// Mitsubishi GX Works2 project: automation_group14_plc_280124   PLC: FX3G

// global labels: Global1
VAR_GLOBAL
  start AT X007 : BOOL;
  During_day AT Y007 : BOOL;
  Emergency_B AT X011 : BOOL;
  Analog_Input1 AT D8280 : INT;
  input_value AT D8201 : INT;
END_VAR
VAR_GLOBAL CONSTANT
  less_then_5 : REAL;
  check_if_lager : INT := 5;
END_VAR
VAR_GLOBAL
  Lager AT M2 : BOOL;
  On_Switch AT X007 : BOOL;
  analog_output AT D8282 : INT;
  check_inv AT M1 : BOOL;
  Analog_Value1 AT D8288 : INT;
END_VAR
VAR_GLOBAL CONSTANT
  Middle_Val : REAL := 2000;
END_VAR
VAR_GLOBAL
  Beer_Type AT M2 : BOOL;
  enough_inv AT M3 : BOOL;
  check AT Y000 : BOOL;
  Input_val AT D8280 : REAL;
END_VAR
VAR_GLOBAL CONSTANT
  div_by_400 : INT := 400;
END_VAR
VAR_GLOBAL
  save_Analog_V AT D7777 : REAL;
END_VAR
VAR_GLOBAL CONSTANT
  normalization : REAL := 400;
END_VAR
VAR_GLOBAL
  option AT D2000 : REAL;
END_VAR
VAR_GLOBAL CONSTANT
  const_1 : REAL := 5;
END_VAR
VAR_GLOBAL
  inv_good AT M3 : BOOL;
  TC_1 AT Y001 : BOOL;
  TC AT TC1 : BOOL;
END_VAR
VAR_GLOBAL CONSTANT
  timer_1 : REAL := 40;
END_VAR
VAR_GLOBAL
  timer_when_cooking AT TS1 : BOOL;
  y_1 AT Y001 : BOOL;
  TC1 AT TC1 : BOOL;
END_VAR
VAR_GLOBAL CONSTANT
  TIMER_COOKING : INT := 40;
END_VAR
VAR_GLOBAL
  job_1 AT X001 : BOOL;
  lagger_check AT M4 : BOOL;
  pilzner_check AT M5 : BOOL;
END_VAR
VAR_GLOBAL CONSTANT
  Lager_Shmarim_need : REAL := 150;
  Lager_Letet_need : REAL := 12;
  Lager_Kshut_need : REAL := 60;
  Pilzner_Shmarim_need : REAL := 120;
  Pilzner_letet_need : REAL := 6;
  Pilzner_Kshut_need : REAL := 53;
  shmarim : REAL := 301;
  letet : REAL := 200;
  kshut : REAL := 200;
END_VAR
VAR_GLOBAL
  finished_cooking_lagger AT M6 : BOOL;
  shmarim_inv AT D4444 : REAL;
  letet_inv AT D5555 : REAL;
  kshut_inv AT D6666 : REAL;
  finished_cooking_Pilzner AT M7 : BOOL;
  move_to_tsisa AT X005 : BOOL;
  start_tsisa_lagger AT M8 : BOOL;
  start_tsisa_pilzner AT M9 : BOOL;
END_VAR
VAR_GLOBAL CONSTANT
  TValue3 : INT := 30;
END_VAR
VAR_GLOBAL
  TS1 AT TS1 : BOOL;
  Y_3 AT Y003 : BOOL;
  TC_4 AT TC4 : BOOL;
END_VAR
VAR_GLOBAL CONSTANT
  TValue4 : INT := 40;
END_VAR
VAR_GLOBAL
  TS_4 AT TS4 : BOOL;
  y_4 AT Y004 : BOOL;
  X_2 AT X002 : BOOL;
  X_0 AT X000 : BOOL;
  cc_1 AT CC1 : BOOL;
END_VAR
VAR_GLOBAL CONSTANT
  counter5 : INT := 6;
END_VAR
VAR_GLOBAL
  CS_1 AT CS1 : BOOL;
  Y_2 AT Y002 : BOOL;
  m_11 AT M11 : BOOL;
  TC_5 AT TC5 : BOOL;
  TS_5 AT TS5 : BOOL;
  TC_6 AT TC6 : BOOL;
  TS_6 AT TS6 : BOOL;
  m_20 AT M20 : BOOL;
  NumOfPack AT D1111 : REAL;
END_VAR
VAR_GLOBAL CONSTANT
  AddingPack : REAL := 0.1;
END_VAR
VAR_GLOBAL
  DayFinish_Lager AT M18 : BOOL;
  DayFinish_Pilzner AT M19 : BOOL;
END_VAR
VAR_GLOBAL CONSTANT
  MulFourty : REAL := 4000;
END_VAR
VAR_GLOBAL
  m_21 AT M21 : BOOL;
  is_Lager AT M2 : BOOL;
  is_pilzner AT M21 : BOOL;
END_VAR
VAR_GLOBAL CONSTANT
  counter6 : INT := 6;
END_VAR
VAR_GLOBAL
  X0_isOn AT M25 : BOOL;
  DayFinish AT M30 : BOOL;
  Not_day_finish AT M30 : BOOL;
END_VAR
VAR_GLOBAL CONSTANT
  const_2 : REAL := 10;
END_VAR
VAR_GLOBAL
  TC_3 AT TC3 : BOOL;
  TS_3 AT TS3 : BOOL;
  Not_finish_Pack_1 AT M40 : BOOL;
END_VAR
VAR_GLOBAL CONSTANT
  div_forty : REAL := 10;
END_VAR
VAR_GLOBAL
  final_output AT D6000 : REAL;
END_VAR
VAR_GLOBAL CONSTANT
  MulFourty1 : REAL := 10;
END_VAR
VAR_GLOBAL
  analog_output1 AT D8282 : INT;
  TC13 AT TC13 : BOOL;
  TsisaLager AT TC13 : BOOL;
END_VAR
VAR_GLOBAL CONSTANT
  tsisaLager_30 : INT := 30;
END_VAR
VAR_GLOBAL
  TsisaPilzner AT TC14 : BOOL;
END_VAR
VAR_GLOBAL CONSTANT
  tsisaPilzner_40 : INT := 40;
END_VAR
VAR_GLOBAL
  finish_tsia_lager AT TS13 : BOOL;
  finish_tsisa_pilzner AT TS14 : BOOL;
  M_100 AT M100 : BOOL;
  start_blink3 AT TC30 : BOOL;
END_VAR
VAR_GLOBAL CONSTANT
  Blink : INT := 5;
END_VAR
VAR_GLOBAL
  blink_Y3 AT TS30 : BOOL;
  start_blink4 AT TC31 : BOOL;
END_VAR
VAR_GLOBAL CONSTANT
  blink2 : INT := 5;
END_VAR
VAR_GLOBAL
  Blink_Y4 AT TS31 : BOOL;
END_VAR

// task Task_01 (event TRUE, interval 0, priority 31): POU_01

PROGRAM POU_01
(* structured ladder/FBD written out as ST: instructions are called as NAME(EN, inputs, outputs); _pN, _eN, _tN stand for wires *)
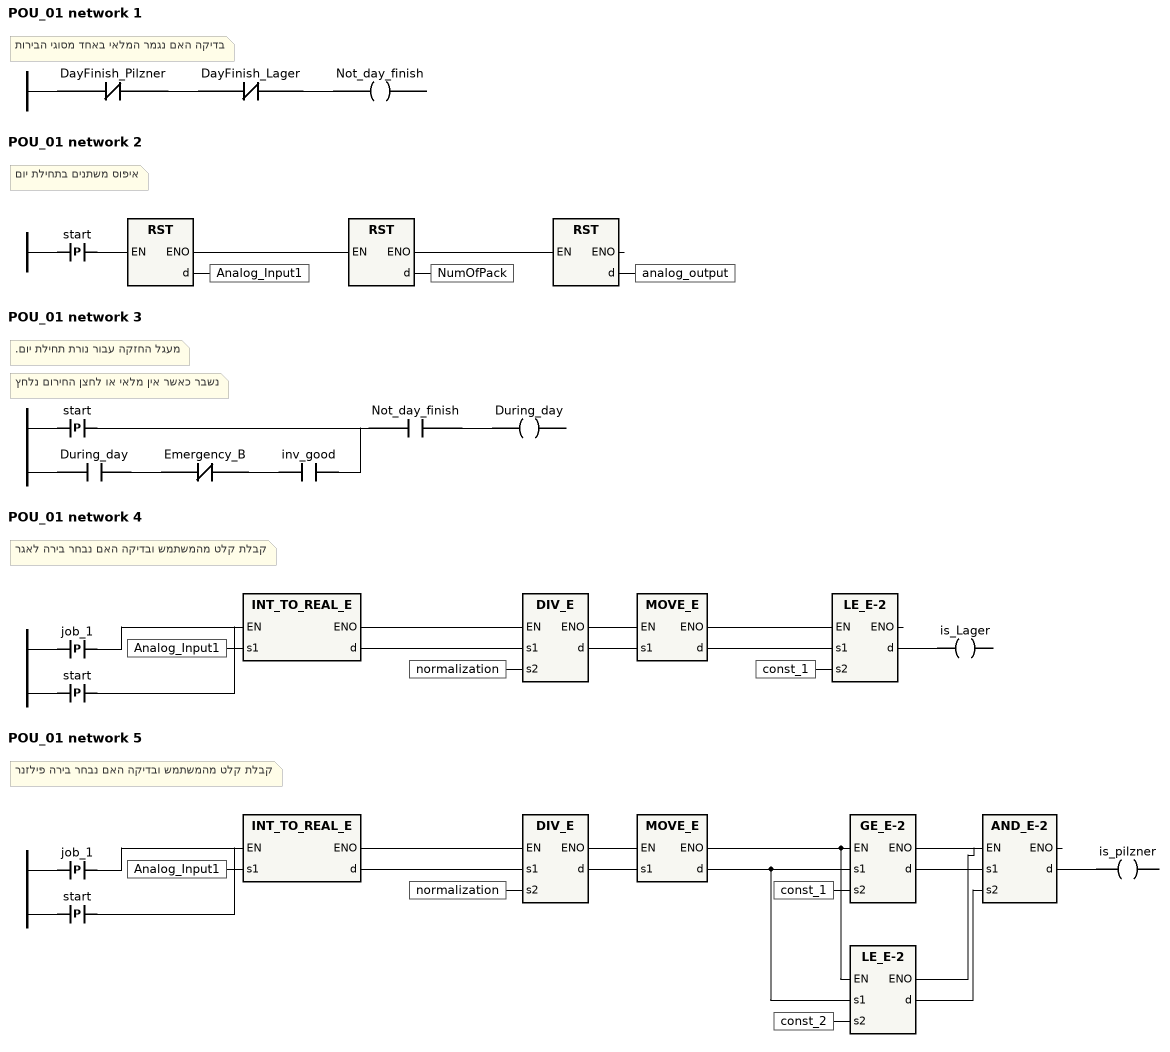
(* network 1 *)
(* בדיקה האם נגמר המלאי באחד מסוגי הבירות *)
Not_day_finish := NOT DayFinish_Pilzner AND NOT DayFinish_Lager;
(* network 2 *)
(* איפוס משתנים בתחילת יום *)
_e1 := RST(LDP(TRUE, start), Analog_Input1);
_e2 := RST(_e1, NumOfPack);
RST(_e2, analog_output);
(* network 3 *)
(* מעגל החזקה עבור נורת תחילת יום. *)
(* נשבר כאשר אין מלאי או לחצן החירום נלחץ *)
During_day := (LDP(TRUE, start) OR (During_day AND NOT Emergency_B AND inv_good)) AND Not_day_finish;
(* network 4 *)
(* קבלת קלט מהמשתמש ובדיקה האם נבחר בירה לאגר *)
_e2 := INT_TO_REAL_E(LDP(TRUE, job_1) OR LDP(TRUE, start), Analog_Input1, _t1);
_e4 := DIV_E(_e2, _t1, normalization, _t3);
_e6 := MOVE_E(_e4, _t3, _t5);
LE_E(_e6, _t5, const_1, _t7);
is_Lager := _t7;
(* network 5 *)
(* קבלת קלט מהמשתמש ובדיקה האם נבחר בירה פילזנר *)
_e2 := INT_TO_REAL_E(LDP(TRUE, job_1) OR LDP(TRUE, start), Analog_Input1, _t1);
_e4 := DIV_E(_e2, _t1, normalization, _t3);
_e6 := MOVE_E(_e4, _t3, _t5);
_e8 := GE_E(_e6, _t5, const_1, _t7);
_e10 := LE_E(_e6, _t5, const_2, _t9);
AND_E(_e8 OR _e10, _t7, _t9, _t11);
is_pilzner := _t11;
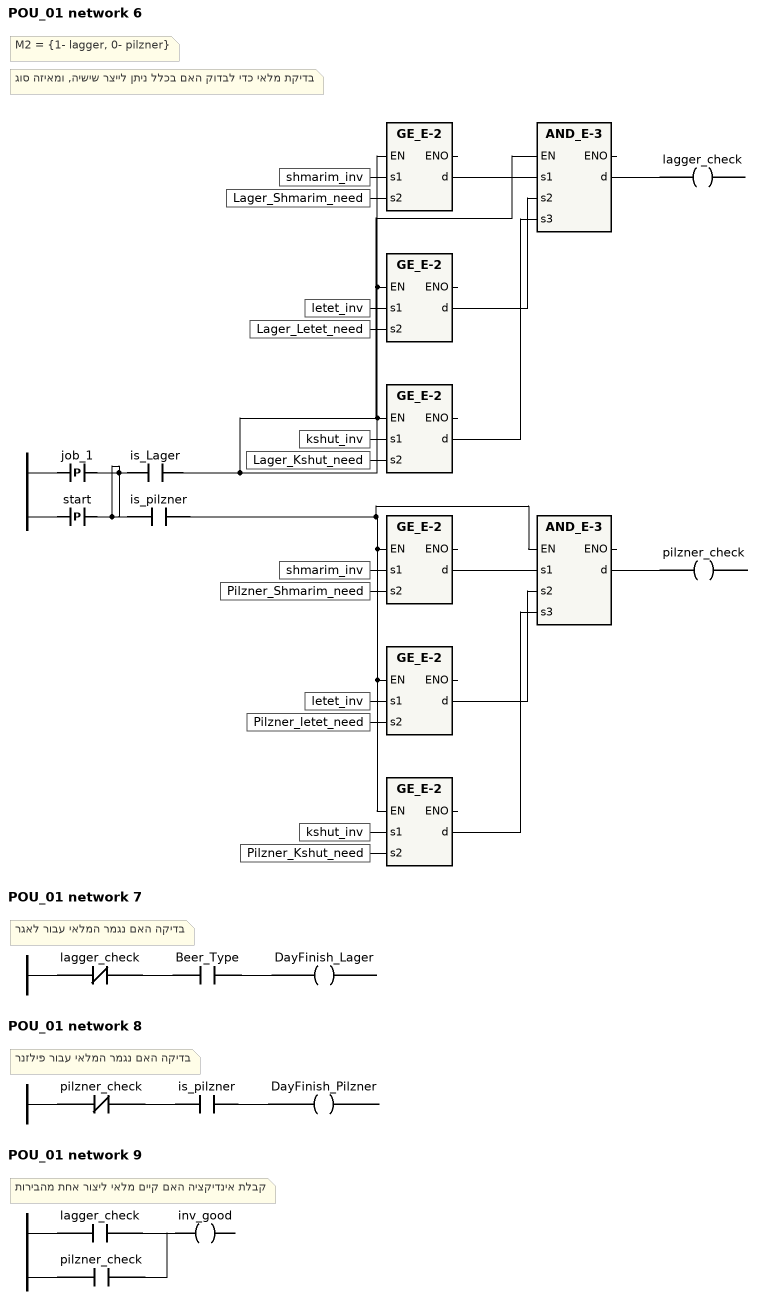
(* network 6 *)
(* M2 = {1- lagger, 0- pilzner} *)
(* בדיקת מלאי כדי לבדוק האם בכלל ניתן לייצר שישיה, ומאיזה סוג *)
_p1 := LDP(TRUE, job_1) OR LDP(TRUE, start);
_p2 := _p1 AND is_Lager;
GE_E(_p2, shmarim_inv, Lager_Shmarim_need, _t3);
GE_E(_p2, letet_inv, Lager_Letet_need, _t4);
GE_E(_p2, kshut_inv, Lager_Kshut_need, _t5);
AND_E(_p2, _t3, _t4, _t5, _t6);
lagger_check := _t6;
_p7 := _p1 AND is_pilzner;
GE_E(_p7, shmarim_inv, Pilzner_Shmarim_need, _t8);
GE_E(_p7, letet_inv, Pilzner_letet_need, _t9);
GE_E(_p7, kshut_inv, Pilzner_Kshut_need, _t10);
AND_E(_p7, _t8, _t9, _t10, _t11);
pilzner_check := _t11;
(* network 7 *)
(* בדיקה האם נגמר המלאי עבור לאגר *)
DayFinish_Lager := NOT lagger_check AND Beer_Type;
(* network 8 *)
(* בדיקה האם נגמר המלאי עבור פילזנר *)
DayFinish_Pilzner := NOT pilzner_check AND is_pilzner;
(* network 9 *)
(* קבלת אינדיקציה האם קיים מלאי ליצור אחת מהבירות *)
inv_good := lagger_check OR pilzner_check;
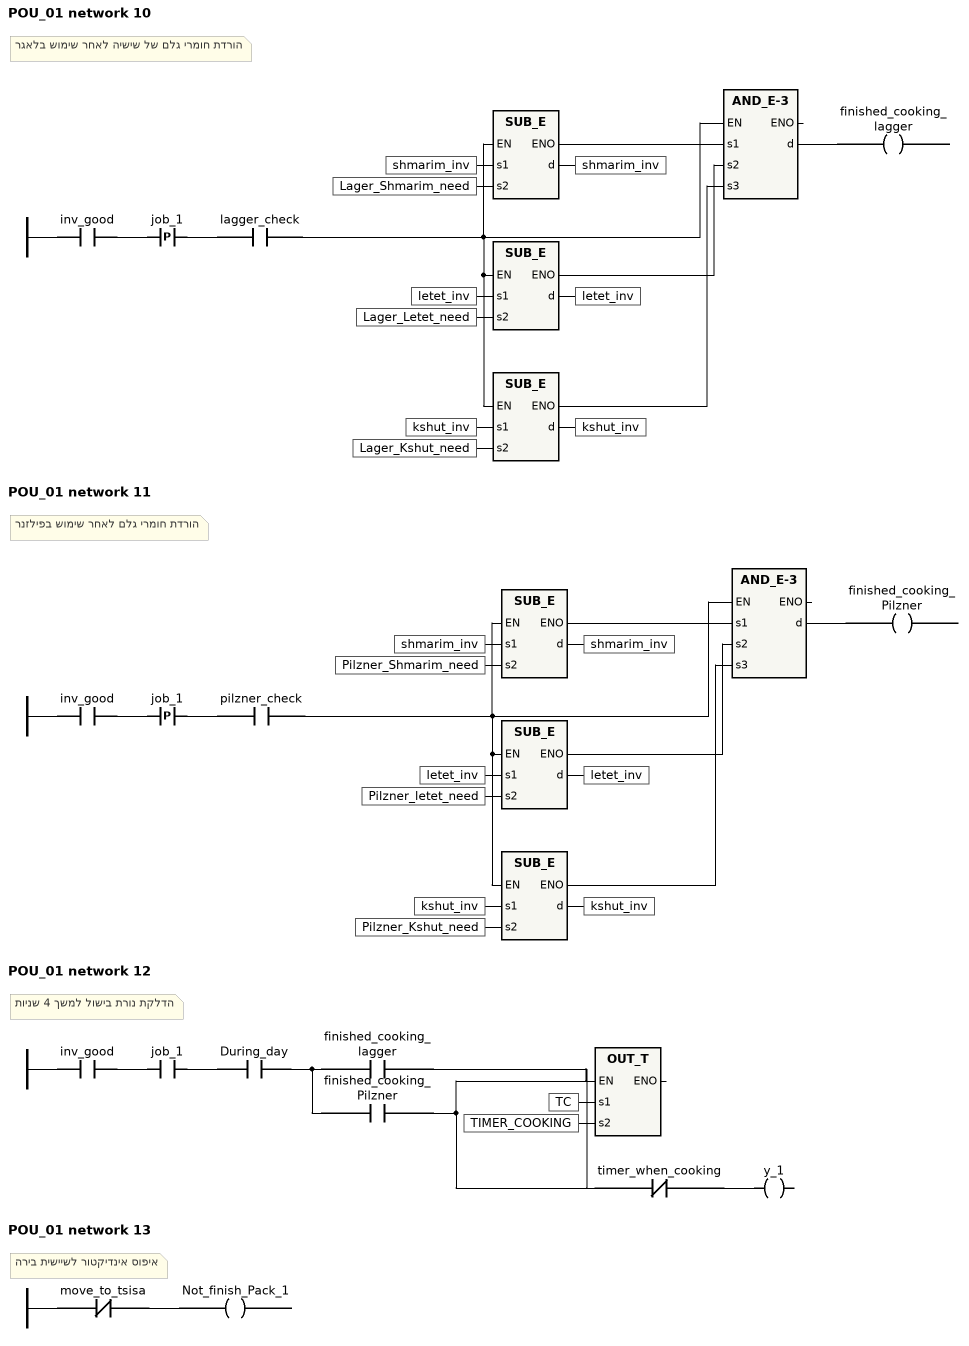
(* network 10 *)
(* הורדת חומרי גלם של שישיה לאחר שימוש בלאגר *)
_p1 := inv_good AND LDP(TRUE, job_1) AND lagger_check;
_e2 := SUB_E(_p1, shmarim_inv, Lager_Shmarim_need, shmarim_inv);
_e3 := SUB_E(_p1, letet_inv, Lager_Letet_need, letet_inv);
_e4 := SUB_E(_p1, kshut_inv, Lager_Kshut_need, kshut_inv);
AND_E(_p1, _e2, _e3, _e4, _t5);
finished_cooking_lagger := _t5;
(* network 11 *)
(* הורדת חומרי גלם לאחר שימוש בפילזנר *)
_p1 := inv_good AND LDP(TRUE, job_1) AND pilzner_check;
_e2 := SUB_E(_p1, shmarim_inv, Pilzner_Shmarim_need, shmarim_inv);
_e3 := SUB_E(_p1, letet_inv, Pilzner_letet_need, letet_inv);
_e4 := SUB_E(_p1, kshut_inv, Pilzner_Kshut_need, kshut_inv);
AND_E(_p1, _e2, _e3, _e4, _t5);
finished_cooking_Pilzner := _t5;
(* network 12 *)
(* הדלקת נורת בישול למשך 4 שניות *)
_p1 := inv_good AND job_1 AND During_day;
_p2 := (_p1 AND finished_cooking_lagger) OR (_p1 AND finished_cooking_Pilzner);
y_1 := _p2 AND NOT timer_when_cooking;
OUT_T(_p2, TC, TIMER_COOKING);
(* network 13 *)
(* איפוס אינדיקטור לשיישית בירה *)
Not_finish_Pack_1 := NOT move_to_tsisa;
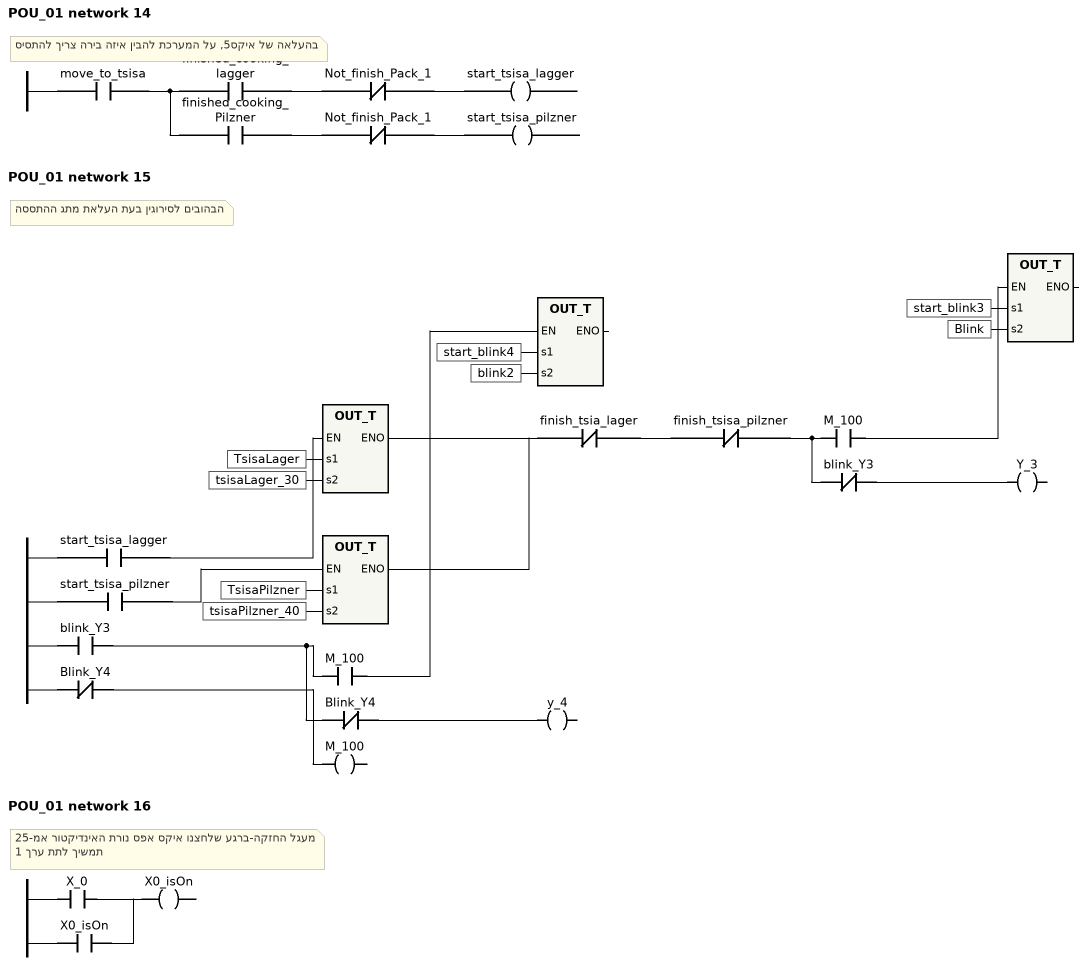
(* network 14 *)
(* בהעלאה של איקס5, על המערכת להבין איזה בירה צריך להתסיס *)
start_tsisa_lagger := move_to_tsisa AND finished_cooking_lagger AND NOT Not_finish_Pack_1;
start_tsisa_pilzner := move_to_tsisa AND finished_cooking_Pilzner AND NOT Not_finish_Pack_1;
(* network 15 *)
(* הבהובים לסירוגין בעת העלאת מתג ההתססה *)
_e1 := OUT_T(start_tsisa_lagger, TsisaLager, tsisaLager_30);
_e2 := OUT_T(start_tsisa_pilzner, TsisaPilzner, tsisaPilzner_40);
_p3 := ((_e1 OR _e2) AND NOT finish_tsia_lager) AND NOT finish_tsisa_pilzner;
OUT_T(_p3 AND M_100, start_blink3, Blink);
Y_3 := _p3 AND NOT blink_Y3;
OUT_T(blink_Y3 AND M_100, start_blink4, blink2);
y_4 := blink_Y3 AND NOT Blink_Y4;
M_100 := NOT Blink_Y4;
(* network 16 *)
(* מעגל החזקה-ברגע שלחצנו איקס אפס נורת האינדיקטור אמ-25 תמשיך לתת ערך 1 *)
X0_isOn := X_0 OR X0_isOn;
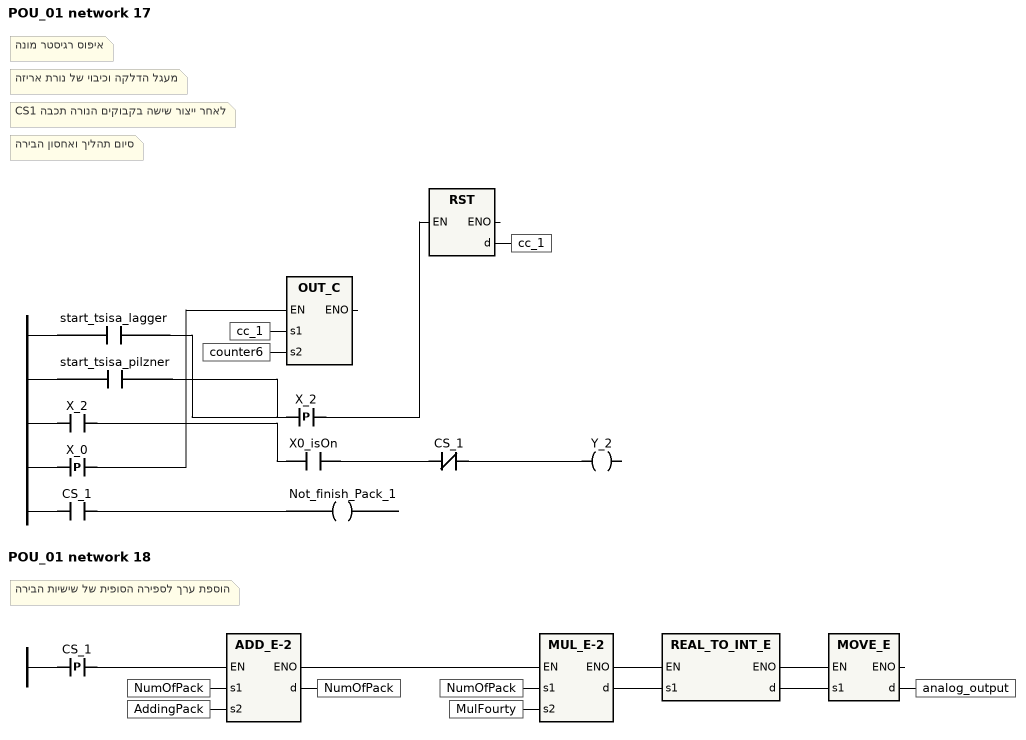
(* network 17 *)
(* איפוס רגיסטר מונה *)
(* מעגל הדלקה וכיבוי של נורת אריזה *)
(* לאחר ייצור שישה בקבוקים הנורה תכבה CS1 *)
(* סיום תהליך ואחסון הבירה *)
RST((start_tsisa_lagger OR start_tsisa_pilzner) AND LDP(TRUE, X_2), cc_1);
Y_2 := X_2 AND X0_isOn AND NOT CS_1;
OUT_C(LDP(TRUE, X_0), cc_1, counter6);
Not_finish_Pack_1 := CS_1;
(* network 18 *)
(* הוספת ערך לספירה הסופית של שישיות הבירה *)
_e1 := ADD_E(LDP(TRUE, CS_1), NumOfPack, AddingPack, NumOfPack);
_e3 := MUL_E(_e1, NumOfPack, MulFourty, _t2);
_e5 := REAL_TO_INT_E(_e3, _t2, _t4);
MOVE_E(_e5, _t4, analog_output);
END_PROGRAM
